FUNCTION_BLOCK EmergencyManagement (* CAT Function Block Type *)
  (* Standard: 61499-2 *)
  (* Version 0.0, 7/4/2026, Schneider Electric, template *)
  PACKAGE SE.Nereda;
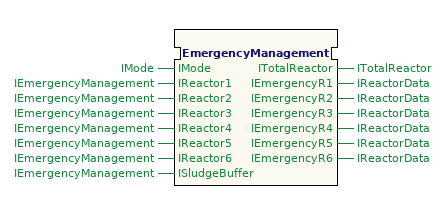
  SOCKETS
    IMode : IMode;
    IReactor1 : IEmergencyManagement;
    IReactor2 : IEmergencyManagement;
    IReactor3 : IEmergencyManagement;
    IReactor4 : IEmergencyManagement;
    IReactor5 : IEmergencyManagement;
    IReactor6 : IEmergencyManagement;
    ISludgeBuffer : IEmergencyManagement;
  END_SOCKETS
  PLUGS
    ITotalReactor : ITotalReactor;
    IEmergencyR1 : IReactorData(pin_7FC77B7D4B4A5A4D := 1);
    IEmergencyR2 : IReactorData(pin_7FC77B7D4B4A5A4D := 2);
    IEmergencyR3 : IReactorData(pin_7FC77B7D4B4A5A4D := 3);
    IEmergencyR4 : IReactorData(pin_7FC77B7D4B4A5A4D := 4);
    IEmergencyR5 : IReactorData(pin_7FC77B7D4B4A5A4D := 5);
    IEmergencyR6 : IReactorData(pin_7FC77B7D4B4A5A4D := 6);
  END_PLUGS
  (* 01 - FUNCTIONNAL INPUT INTERFACE *)
  (* 00 - INITIALIZATION *)
  (* 05 - LOGIC *)
  (* 06 - HMI INTERFACE *)
  (* 03 - FIELD INTERFACE *)
  (* 02 - FUNCTIONNAL OUTPUT INTERFACE *)
  (* Number of Reactors Exist *)
  (* 04 - CHILDREN *)
  (* 4A - TYPICALS *)
  (* Actual Cycle Time (CT_reactor_actual) CT_ReactorActual = (N_AvailableReactors / N_TotalReactors) x CT_Nominal *)
  (* Next Feed Horizon Calculation (Scheduler) *)
  (* Emergency ON *)
  (* Number of Reactors Available *)
  (* Start Feed Position *)
  (* Feed Interval (Start_IntervalV = CT_ReactorActual / N_AvailableReactors) *)
  (* Emergency Reactors Control (Start & Stop) *)
  (* Time Sice Start Feed *)
  (* Emergency Initialization *)
  (* Start Feed Position This functional block manages the reactor position order, which determines the sequence in which the feeds are started. We request an update of the "Reactor To Start Feed" position in the following two cases: - In the logic that controls the start of the Emergency Recipe Sequence. - In the update performed after the start of each feed. *)
  (* Comment These function blocks (`SD_WS2_Initialization_Manager` and `RxNoAvThenRxAv`) must be modified to match the number of reactors in your plant. *)
  FBS
    INIT : plcStart(Prio := 50, Delay := T#0ms);
    NumberOfReactors : ADD_196CF02D1C6422644; {SET_ATTRIBUTE(Configuration.GenericFBType.InterfaceParams, Runtime.Standard#CNT:=6;IN${CNT$}:LREAL)}
    IThis : EmergencyManagement_HMI(QI := TRUE);
    SmoothNumberOfReactors : LRealValueChanged;
    SmoothNumberOfReactors1 : LREAL2REAL;
    CT_ReactorActual : CT_ReactorActual;
    SmoothCT_ReactorActual : RealValueChanged;
    EmergencyON : COMPARE_739E3FB559152FE(IN2 := 3); {SET_ATTRIBUTE(Configuration.GenericFBType.InterfaceParams, Runtime.Standard#CNT:=2;IN${CNT$}:INT)}
    SmoothEmergencyON : boolValueChanged;
    NumberOfReactorsAv : ADD_196CF02D1C6422644; {SET_ATTRIBUTE(Configuration.GenericFBType.InterfaceParams, Runtime.Standard#CNT:=6;IN${CNT$}:LREAL)}
    SmoothNumberOfReactorsAv : LRealValueChanged;
    NumberOfReactorsAv2 : LREAL2REAL;
    BOOL2INT : BOOL2INT_6;
    StartFeedPosition : StartFeedPosition;
    SmoothNumberOfReactors2 : REAL2INT;
    ReactorFeedInterval : StartIntervalCalc;
    EmergencyReactorsControl : EmergencyManagementControl;
    NumberOfReactorsAv3 : REAL2INT;
    StartUpDelay : E_DELAY_V_D;
    Retrigger_StartFeedPosition : RetriggerEvent(pin_CFF51EFF0A91DC53 := 3, pin_FDD5DC24A8674AF6 := T#1s);
    ForceAvaibility : ReactorAvCtrl;
    SmoothFeedInterval : RealValueChanged;
    TimeSinceStartFeedR1 : RealValueChanged;
    TimeSinceStartFeedR2 : RealValueChanged;
    TimeSinceStartFeedR3 : RealValueChanged;
    TimeSinceStartFeedR4 : RealValueChanged;
    TimeSinceStartFeedR5 : RealValueChanged;
    TimeSinceStartFeedR6 : RealValueChanged;
    NextFeedHorizon : NextFeedHorizon;
    BOOL2INT1 : BOOL2INT_6;
    FeedRun : E_PERMIT;
    FeedStarted : OR_65BD917F4F2EC165; {SET_ATTRIBUTE(Configuration.GenericFBType.InterfaceParams, Runtime.Standard#CNT:=6;OUT:BOOL)}
    FeedCmdTimeOutR1 : TimeOut(pin_5F65B6CE2660F5EB := T#500ms);
    FeedCmdTimeOutR2 : TimeOut(pin_5F65B6CE2660F5EB := T#500ms);
    FeedCmdTimeOutR3 : TimeOut(pin_5F65B6CE2660F5EB := T#500ms);
    FeedCmdTimeOutR4 : TimeOut(pin_5F65B6CE2660F5EB := T#500ms);
    FeedCmdTimeOutR5 : TimeOut(pin_5F65B6CE2660F5EB := T#500ms);
    FeedCmdTimeOutR6 : TimeOut(pin_5F65B6CE2660F5EB := T#500ms);
    SD_WS2_Initialization_Manager : SDInitDone(pin_9BB0B293AF87503A := TRUE, pin_46B4EB9EBD3AAF12 := TRUE, pin_7A6A945A02239988 := TRUE);
    Wait : E_DELAY(DT := T#500ms);
    UPDATE_POS : E_DELAY(DT := T#1s);
    Delay : E_DELAY_V_D(DT1 := T#2s);
    FeedStartedSmooth : BoolValueChanged_6;
    ReactorAvaibilityChanged : BoolValueChanged_6;
    UPDATE_POS_EO : E_MERGE;
    EmergencyONPermit : E_PERMIT;
    RxNoAvThenRxAv : RNoAvThenRAv(pin_F258A2B490CD5DB0 := TRUE, pin_1987E369E19A00E5 := TRUE, pin_36BA10F8F7A678CF := TRUE);
    Wait1 : E_DELAY(DT := T#500ms);
  END_FBS
  EVENT_CONNECTIONS
    EmergencyON.CNF TO SmoothEmergencyON.REQ;
    IMode.MODE TO EmergencyON.REQ;
    IMode.MODE TO EmergencyReactorsControl.57E2081A00120193;
    IReactor2.PHASE_NO_ABORTED TO ForceAvaibility.AA8C7A967C5CED2A;
    IReactor2.PHASE_NO_ABORTED TO EmergencyReactorsControl.FC096638C9B2EBE7;
    IReactor2.FEED_TIME TO StartFeedPosition.9A3C6DCF3E2E1FB0;
    IReactor2.12FB600C11F75EA2 TO StartFeedPosition.9A3C6DCF3E2E1FB0;
    IReactor2.12FB600C11F75EA2 TO EmergencyReactorsControl.3FB25A98F6D2D397;
    IReactor2.12FB600C11F75EA2 TO EmergencyReactorsControl.FC096638C9B2EBE7;
    StartUpDelay.INITO TO IReactor2.33EC5B834E8FFAF3;
    IReactor1.PHASE_NO_ABORTED TO ForceAvaibility.AA8C7A967C5CED2A;
    IReactor1.PHASE_NO_ABORTED TO EmergencyReactorsControl.FC096638C9B2EBE7;
    IReactor1.FEED_TIME TO StartFeedPosition.9A3C6DCF3E2E1FB0;
    IReactor1.12FB600C11F75EA2 TO StartFeedPosition.9A3C6DCF3E2E1FB0;
    IReactor1.12FB600C11F75EA2 TO EmergencyReactorsControl.3FB25A98F6D2D397;
    IReactor1.12FB600C11F75EA2 TO EmergencyReactorsControl.FC096638C9B2EBE7;
    StartUpDelay.INITO TO IReactor1.33EC5B834E8FFAF3;
    StartUpDelay.INITO TO IReactor3.33EC5B834E8FFAF3;
    IReactor3.PHASE_NO_ABORTED TO ForceAvaibility.AA8C7A967C5CED2A;
    IReactor3.PHASE_NO_ABORTED TO EmergencyReactorsControl.FC096638C9B2EBE7;
    IReactor3.FEED_TIME TO StartFeedPosition.9A3C6DCF3E2E1FB0;
    IReactor3.12FB600C11F75EA2 TO StartFeedPosition.9A3C6DCF3E2E1FB0;
    IReactor3.12FB600C11F75EA2 TO EmergencyReactorsControl.3FB25A98F6D2D397;
    IReactor3.12FB600C11F75EA2 TO EmergencyReactorsControl.FC096638C9B2EBE7;
    StartUpDelay.INITO TO IReactor4.33EC5B834E8FFAF3;
    IReactor4.PHASE_NO_ABORTED TO ForceAvaibility.AA8C7A967C5CED2A;
    IReactor4.PHASE_NO_ABORTED TO EmergencyReactorsControl.FC096638C9B2EBE7;
    IReactor4.FEED_TIME TO StartFeedPosition.9A3C6DCF3E2E1FB0;
    IReactor4.12FB600C11F75EA2 TO StartFeedPosition.9A3C6DCF3E2E1FB0;
    IReactor4.12FB600C11F75EA2 TO EmergencyReactorsControl.3FB25A98F6D2D397;
    IReactor4.12FB600C11F75EA2 TO EmergencyReactorsControl.FC096638C9B2EBE7;
    StartUpDelay.INITO TO IReactor5.33EC5B834E8FFAF3;
    IReactor5.PHASE_NO_ABORTED TO ForceAvaibility.AA8C7A967C5CED2A;
    IReactor5.PHASE_NO_ABORTED TO EmergencyReactorsControl.FC096638C9B2EBE7;
    IReactor5.FEED_TIME TO StartFeedPosition.9A3C6DCF3E2E1FB0;
    IReactor5.12FB600C11F75EA2 TO StartFeedPosition.9A3C6DCF3E2E1FB0;
    IReactor5.12FB600C11F75EA2 TO EmergencyReactorsControl.3FB25A98F6D2D397;
    IReactor5.12FB600C11F75EA2 TO EmergencyReactorsControl.FC096638C9B2EBE7;
    IReactor6.PHASE_NO_ABORTED TO ForceAvaibility.AA8C7A967C5CED2A;
    IReactor6.PHASE_NO_ABORTED TO EmergencyReactorsControl.FC096638C9B2EBE7;
    IReactor6.FEED_TIME TO StartFeedPosition.9A3C6DCF3E2E1FB0;
    IReactor6.12FB600C11F75EA2 TO StartFeedPosition.9A3C6DCF3E2E1FB0;
    IReactor6.12FB600C11F75EA2 TO EmergencyReactorsControl.3FB25A98F6D2D397;
    IReactor6.12FB600C11F75EA2 TO EmergencyReactorsControl.FC096638C9B2EBE7;
    StartUpDelay.INITO TO IReactor6.33EC5B834E8FFAF3;
    SmoothNumberOfReactors2.6FC99A5BD1C38561 TO EmergencyReactorsControl.3FB25A98F6D2D397;
    NumberOfReactorsAv3.6FC99A5BD1C38561 TO EmergencyReactorsControl.FC096638C9B2EBE7;
    StartUpDelay.1457E63E0C241C83 TO EmergencyReactorsControl.B99EA0FFDDD9DD73;
    EmergencyReactorsControl.5425B5FF7C2B3EA7 TO IEmergencyR1.395F2A7D1AB6A478;
    EmergencyReactorsControl.5425B5FF7C2B3EA7 TO IEmergencyR2.395F2A7D1AB6A478;
    EmergencyReactorsControl.5425B5FF7C2B3EA7 TO IEmergencyR4.395F2A7D1AB6A478;
    EmergencyReactorsControl.5425B5FF7C2B3EA7 TO IEmergencyR3.395F2A7D1AB6A478;
    EmergencyReactorsControl.5425B5FF7C2B3EA7 TO IEmergencyR5.395F2A7D1AB6A478;
    EmergencyReactorsControl.5425B5FF7C2B3EA7 TO IEmergencyR6.395F2A7D1AB6A478;
    EmergencyReactorsControl.B331D681195361F6 TO StartUpDelay.START;
    StartUpDelay.INITO TO ForceAvaibility.227A3F3489EABE9B;
    SmoothNumberOfReactors2.6FC99A5BD1C38561 TO ITotalReactor.TOTAL_REACTOR;
    SmoothEmergencyON.CHD TO IEmergencyR1.E1D373823D64ACA0;
    SmoothEmergencyON.CHD TO IEmergencyR2.E1D373823D64ACA0;
    SmoothEmergencyON.CHD TO IEmergencyR3.E1D373823D64ACA0;
    SmoothEmergencyON.CHD TO IEmergencyR4.E1D373823D64ACA0;
    SmoothEmergencyON.CHD TO IEmergencyR5.E1D373823D64ACA0;
    SmoothEmergencyON.CHD TO IEmergencyR6.E1D373823D64ACA0;
    NumberOfReactors.CNF TO SmoothNumberOfReactors.77F8F9CFF707DAFF;
    SmoothNumberOfReactors.93AE3729A9342678 TO SmoothNumberOfReactors1.DD5870AA881150BB;
    SmoothNumberOfReactors1.6FC99A5BD1C38561 TO SmoothNumberOfReactors2.DD5870AA881150BB;
    SmoothNumberOfReactors2.6FC99A5BD1C38561 TO CT_ReactorActual.B5AD92DA165DFC02;
    BOOL2INT.6FC99A5BD1C38561 TO NumberOfReactorsAv.REQ;
    NumberOfReactorsAv.CNF TO SmoothNumberOfReactorsAv.77F8F9CFF707DAFF;
    SmoothNumberOfReactorsAv.93AE3729A9342678 TO NumberOfReactorsAv2.DD5870AA881150BB;
    NumberOfReactorsAv2.6FC99A5BD1C38561 TO NumberOfReactorsAv3.DD5870AA881150BB;
    NumberOfReactorsAv3.6FC99A5BD1C38561 TO CT_ReactorActual.B5AD92DA165DFC02;
    NumberOfReactorsAv3.6FC99A5BD1C38561 TO ReactorFeedInterval.56116EFC174D2765;
    CT_ReactorActual.FB6D4D448571E6B8 TO SmoothCT_ReactorActual.77F8F9CFF707DAFF;
    SmoothCT_ReactorActual.93AE3729A9342678 TO ReactorFeedInterval.56116EFC174D2765;
    EmergencyReactorsControl.4DD14AD6E2842102 TO StartFeedPosition.DD2DDDBAAA645E47;
    SmoothNumberOfReactorsAv.350834820611931F TO StartFeedPosition.9A3C6DCF3E2E1FB0;
    Retrigger_StartFeedPosition.4002AEF0814D09CF TO EmergencyReactorsControl.7CCC917F1D2D8CDF;
    SmoothCT_ReactorActual.93AE3729A9342678 TO IEmergencyR1.198EF041C70827BC;
    SmoothCT_ReactorActual.93AE3729A9342678 TO IEmergencyR2.198EF041C70827BC;
    SmoothCT_ReactorActual.93AE3729A9342678 TO IEmergencyR3.198EF041C70827BC;
    SmoothCT_ReactorActual.93AE3729A9342678 TO IEmergencyR4.198EF041C70827BC;
    SmoothCT_ReactorActual.93AE3729A9342678 TO IEmergencyR5.198EF041C70827BC;
    SmoothCT_ReactorActual.93AE3729A9342678 TO IEmergencyR6.198EF041C70827BC;
    SmoothFeedInterval.93AE3729A9342678 TO IEmergencyR1.9D1E5F7369C5538B;
    SmoothFeedInterval.93AE3729A9342678 TO IEmergencyR2.9D1E5F7369C5538B;
    SmoothFeedInterval.93AE3729A9342678 TO IEmergencyR3.9D1E5F7369C5538B;
    SmoothFeedInterval.93AE3729A9342678 TO IEmergencyR4.9D1E5F7369C5538B;
    SmoothFeedInterval.93AE3729A9342678 TO IEmergencyR5.9D1E5F7369C5538B;
    SmoothFeedInterval.93AE3729A9342678 TO IEmergencyR6.9D1E5F7369C5538B;
    EmergencyReactorsControl.E01285EC1A4C329B TO IEmergencyR1.61CD32E3E6AEDF7D;
    EmergencyReactorsControl.E01285EC1A4C329B TO IEmergencyR2.61CD32E3E6AEDF7D;
    EmergencyReactorsControl.E01285EC1A4C329B TO IEmergencyR3.61CD32E3E6AEDF7D;
    EmergencyReactorsControl.E01285EC1A4C329B TO IEmergencyR4.61CD32E3E6AEDF7D;
    EmergencyReactorsControl.E01285EC1A4C329B TO IEmergencyR5.61CD32E3E6AEDF7D;
    EmergencyReactorsControl.E01285EC1A4C329B TO IEmergencyR6.61CD32E3E6AEDF7D;
    Retrigger_StartFeedPosition.4002AEF0814D09CF TO IEmergencyR1.911F6EFE27823BFD;
    Retrigger_StartFeedPosition.4002AEF0814D09CF TO IEmergencyR2.911F6EFE27823BFD;
    Retrigger_StartFeedPosition.4002AEF0814D09CF TO IEmergencyR3.911F6EFE27823BFD;
    Retrigger_StartFeedPosition.4002AEF0814D09CF TO IEmergencyR4.911F6EFE27823BFD;
    Retrigger_StartFeedPosition.4002AEF0814D09CF TO IEmergencyR5.911F6EFE27823BFD;
    Retrigger_StartFeedPosition.4002AEF0814D09CF TO IEmergencyR6.911F6EFE27823BFD;
    ForceAvaibility.A1ADA5210E38DA8E TO BOOL2INT.DD5870AA881150BB;
    ForceAvaibility.8EE38BB13A892011 TO NextFeedHorizon.E161DD05340F6BD8;
    ReactorFeedInterval.8A437FBF24BFC92F TO SmoothFeedInterval.77F8F9CFF707DAFF;
    EmergencyReactorsControl.BDC96AACAB3D2769 TO IEmergencyR1.1C1DD8946F24CFF9;
    EmergencyReactorsControl.BDC96AACAB3D2769 TO IEmergencyR2.1C1DD8946F24CFF9;
    EmergencyReactorsControl.BDC96AACAB3D2769 TO IEmergencyR3.1C1DD8946F24CFF9;
    EmergencyReactorsControl.BDC96AACAB3D2769 TO IEmergencyR4.1C1DD8946F24CFF9;
    EmergencyReactorsControl.BDC96AACAB3D2769 TO IEmergencyR5.1C1DD8946F24CFF9;
    EmergencyReactorsControl.BDC96AACAB3D2769 TO IEmergencyR6.1C1DD8946F24CFF9;
    IReactor1.FEED_TIME TO TimeSinceStartFeedR1.77F8F9CFF707DAFF;
    IReactor2.FEED_TIME TO TimeSinceStartFeedR1.77F8F9CFF707DAFF;
    IReactor3.FEED_TIME TO TimeSinceStartFeedR1.77F8F9CFF707DAFF;
    IReactor4.FEED_TIME TO TimeSinceStartFeedR1.77F8F9CFF707DAFF;
    IReactor5.FEED_TIME TO TimeSinceStartFeedR1.77F8F9CFF707DAFF;
    IReactor6.FEED_TIME TO TimeSinceStartFeedR1.77F8F9CFF707DAFF;
    TimeSinceStartFeedR1.350834820611931F TO TimeSinceStartFeedR2.77F8F9CFF707DAFF;
    TimeSinceStartFeedR2.350834820611931F TO TimeSinceStartFeedR3.77F8F9CFF707DAFF;
    TimeSinceStartFeedR4.350834820611931F TO TimeSinceStartFeedR5.77F8F9CFF707DAFF;
    TimeSinceStartFeedR5.350834820611931F TO TimeSinceStartFeedR6.77F8F9CFF707DAFF;
    TimeSinceStartFeedR3.350834820611931F TO TimeSinceStartFeedR4.77F8F9CFF707DAFF;
    NextFeedHorizon.D6F8783AE30F537C TO Delay.INIT;
    SmoothFeedInterval.93AE3729A9342678 TO NextFeedHorizon.7F05D9AA837FB21B;
    TimeSinceStartFeedR1.93AE3729A9342678 TO NextFeedHorizon.7F05D9AA837FB21B;
    TimeSinceStartFeedR2.93AE3729A9342678 TO NextFeedHorizon.7F05D9AA837FB21B;
    TimeSinceStartFeedR3.93AE3729A9342678 TO NextFeedHorizon.7F05D9AA837FB21B;
    TimeSinceStartFeedR4.93AE3729A9342678 TO NextFeedHorizon.7F05D9AA837FB21B;
    TimeSinceStartFeedR5.93AE3729A9342678 TO NextFeedHorizon.7F05D9AA837FB21B;
    TimeSinceStartFeedR6.93AE3729A9342678 TO NextFeedHorizon.7F05D9AA837FB21B;
    Retrigger_StartFeedPosition.4002AEF0814D09CF TO NextFeedHorizon.7F05D9AA837FB21B;
    NumberOfReactorsAv3.6FC99A5BD1C38561 TO NextFeedHorizon.7F05D9AA837FB21B;
    SmoothNumberOfReactors2.6FC99A5BD1C38561 TO NextFeedHorizon.7F05D9AA837FB21B;
    IReactor1.12FB600C11F75EA2 TO BOOL2INT1.DD5870AA881150BB;
    IReactor2.12FB600C11F75EA2 TO BOOL2INT1.DD5870AA881150BB;
    IReactor3.12FB600C11F75EA2 TO BOOL2INT1.DD5870AA881150BB;
    IReactor4.12FB600C11F75EA2 TO BOOL2INT1.DD5870AA881150BB;
    IReactor5.12FB600C11F75EA2 TO BOOL2INT1.DD5870AA881150BB;
    IReactor6.12FB600C11F75EA2 TO BOOL2INT1.DD5870AA881150BB;
    BOOL2INT1.6FC99A5BD1C38561 TO NumberOfReactors.REQ;
    NextFeedHorizon.A8C1183CD65D2C2F TO EmergencyReactorsControl.F396AB99E066BF1B;
    NextFeedHorizon.3C658083FB00E376 TO EmergencyReactorsControl.EE2641E02BEB131E;
    ForceAvaibility.D789D01B8B35E207 TO IEmergencyR1.7D5F3067068DE334;
    ForceAvaibility.D789D01B8B35E207 TO IEmergencyR2.7D5F3067068DE334;
    ForceAvaibility.D789D01B8B35E207 TO IEmergencyR3.7D5F3067068DE334;
    ForceAvaibility.D789D01B8B35E207 TO IEmergencyR4.7D5F3067068DE334;
    ForceAvaibility.D789D01B8B35E207 TO IEmergencyR5.7D5F3067068DE334;
    ForceAvaibility.D789D01B8B35E207 TO IEmergencyR6.7D5F3067068DE334;
    INIT.FIRST_INIT TO IThis.11B0EEC0AF1F6F5A;
    INIT.REDO_INIT TO IThis.11B0EEC0AF1F6F5A;
    Retrigger_StartFeedPosition.4002AEF0814D09CF TO IThis.6A631B6723098E8B;
    IEmergencyR1.D499D06F1953A020 TO IThis.6A631B6723098E8B;
    IReactor1.FEED_TIME TO IThis.6A631B6723098E8B;
    Retrigger_StartFeedPosition.4002AEF0814D09CF TO IThis.662D34935A18D4C8;
    IEmergencyR2.D499D06F1953A020 TO IThis.662D34935A18D4C8;
    IReactor2.FEED_TIME TO IThis.662D34935A18D4C8;
    IReactor3.FEED_TIME TO IThis.D5FE897AB4BE07D5;
    Retrigger_StartFeedPosition.4002AEF0814D09CF TO IThis.D5FE897AB4BE07D5;
    IEmergencyR3.D499D06F1953A020 TO IThis.D5FE897AB4BE07D5;
    Retrigger_StartFeedPosition.4002AEF0814D09CF TO IThis.0FC97BC77AEF2FB1;
    IEmergencyR4.D499D06F1953A020 TO IThis.0FC97BC77AEF2FB1;
    Retrigger_StartFeedPosition.4002AEF0814D09CF TO IThis.AD50BDBEE1844666;
    IEmergencyR5.D499D06F1953A020 TO IThis.AD50BDBEE1844666;
    Retrigger_StartFeedPosition.4002AEF0814D09CF TO IThis.883D86C4850F1B98;
    IEmergencyR6.D499D06F1953A020 TO IThis.883D86C4850F1B98;
    SmoothCT_ReactorActual.93AE3729A9342678 TO IThis.BCC6AEC920D25E91;
    IThis.B3B324179F7F1286 TO IThis.6FE84D876AB4D285;
    SmoothNumberOfReactors2.6FC99A5BD1C38561 TO IThis.6FE84D876AB4D285;
    NumberOfReactorsAv3.6FC99A5BD1C38561 TO IThis.6FE84D876AB4D285;
    SmoothFeedInterval.93AE3729A9342678 TO IThis.FF5508DDAEC8BEFB;
    EmergencyReactorsControl.57B86B24E58CE6DD TO IThis.C9F34726889CA7BE;
    SmoothEmergencyON.CHD TO IThis.9D03013895CCEF05;
    StartUpDelay.INITO TO IThis.32376FF6F2E25CA6;
    IThis.69E91E9E46EEE4A5 TO StartUpDelay.INIT;
    IThis.B3B324179F7F1286 TO CT_ReactorActual.B5AD92DA165DFC02;
    IThis.13B659E2726FB2AF TO StartUpDelay.8C325F07198FCB13;
    IReactor4.FEED_TIME TO IThis.0FC97BC77AEF2FB1;
    IReactor5.FEED_TIME TO IThis.AD50BDBEE1844666;
    IReactor6.FEED_TIME TO IThis.883D86C4850F1B98;
    NextFeedHorizon.5939463105CA5EBC TO IEmergencyR1.B3BDDBF095B97A2B;
    NextFeedHorizon.5939463105CA5EBC TO IEmergencyR2.B3BDDBF095B97A2B;
    NextFeedHorizon.5939463105CA5EBC TO IEmergencyR3.B3BDDBF095B97A2B;
    NextFeedHorizon.5939463105CA5EBC TO IEmergencyR4.B3BDDBF095B97A2B;
    NextFeedHorizon.5939463105CA5EBC TO IEmergencyR5.B3BDDBF095B97A2B;
    NextFeedHorizon.5939463105CA5EBC TO IEmergencyR6.B3BDDBF095B97A2B;
    FeedStarted.CNF TO FeedRun.EI;
    IEmergencyR1.138EEC247A2C05E7 TO FeedStartedSmooth.77F8F9CFF707DAFF;
    IEmergencyR2.138EEC247A2C05E7 TO FeedStartedSmooth.77F8F9CFF707DAFF;
    IEmergencyR3.138EEC247A2C05E7 TO FeedStartedSmooth.77F8F9CFF707DAFF;
    IEmergencyR4.138EEC247A2C05E7 TO FeedStartedSmooth.77F8F9CFF707DAFF;
    IEmergencyR5.138EEC247A2C05E7 TO FeedStartedSmooth.77F8F9CFF707DAFF;
    IEmergencyR6.138EEC247A2C05E7 TO FeedStartedSmooth.77F8F9CFF707DAFF;
    EmergencyReactorsControl.6CCD34FECBD70B12 TO StartUpDelay.STOP;
    FeedCmdTimeOutR1.A86E94B0584B0184 TO IEmergencyR1.395F2A7D1AB6A478;
    FeedCmdTimeOutR2.A86E94B0584B0184 TO IEmergencyR2.395F2A7D1AB6A478;
    FeedCmdTimeOutR3.A86E94B0584B0184 TO IEmergencyR3.395F2A7D1AB6A478;
    FeedCmdTimeOutR4.A86E94B0584B0184 TO IEmergencyR4.395F2A7D1AB6A478;
    FeedCmdTimeOutR5.A86E94B0584B0184 TO IEmergencyR5.395F2A7D1AB6A478;
    FeedCmdTimeOutR6.A86E94B0584B0184 TO IEmergencyR6.395F2A7D1AB6A478;
    EmergencyReactorsControl.5425B5FF7C2B3EA7 TO FeedCmdTimeOutR1.C17BD4ED345C3B34;
    EmergencyReactorsControl.5425B5FF7C2B3EA7 TO FeedCmdTimeOutR2.C17BD4ED345C3B34;
    EmergencyReactorsControl.5425B5FF7C2B3EA7 TO FeedCmdTimeOutR3.C17BD4ED345C3B34;
    EmergencyReactorsControl.5425B5FF7C2B3EA7 TO FeedCmdTimeOutR4.C17BD4ED345C3B34;
    EmergencyReactorsControl.5425B5FF7C2B3EA7 TO FeedCmdTimeOutR5.C17BD4ED345C3B34;
    EmergencyReactorsControl.5425B5FF7C2B3EA7 TO FeedCmdTimeOutR6.C17BD4ED345C3B34;
    IEmergencyR1.138EEC247A2C05E7 TO FeedCmdTimeOutR1.99EC5987D752BADB;
    IEmergencyR2.138EEC247A2C05E7 TO FeedCmdTimeOutR2.99EC5987D752BADB;
    IEmergencyR3.138EEC247A2C05E7 TO FeedCmdTimeOutR3.99EC5987D752BADB;
    IEmergencyR4.138EEC247A2C05E7 TO FeedCmdTimeOutR4.99EC5987D752BADB;
    IEmergencyR5.138EEC247A2C05E7 TO FeedCmdTimeOutR5.99EC5987D752BADB;
    IEmergencyR6.138EEC247A2C05E7 TO FeedCmdTimeOutR6.99EC5987D752BADB;
    NextFeedHorizon.D6F8783AE30F537C TO IEmergencyR1.CF316F4BA7C11A07;
    NextFeedHorizon.D6F8783AE30F537C TO IEmergencyR2.CF316F4BA7C11A07;
    NextFeedHorizon.D6F8783AE30F537C TO IEmergencyR3.CF316F4BA7C11A07;
    NextFeedHorizon.D6F8783AE30F537C TO IEmergencyR4.CF316F4BA7C11A07;
    NextFeedHorizon.D6F8783AE30F537C TO IEmergencyR5.CF316F4BA7C11A07;
    NextFeedHorizon.D6F8783AE30F537C TO IEmergencyR6.CF316F4BA7C11A07;
    EmergencyReactorsControl.E01285EC1A4C329B TO SD_WS2_Initialization_Manager.B4ABE90B67562793;
    SmoothEmergencyON.CHD TO SD_WS2_Initialization_Manager.08F744362D65AFEF;
    SD_WS2_Initialization_Manager.349B3D6587A5C960 TO IEmergencyR1.77175193A5DFB16A;
    SD_WS2_Initialization_Manager.349B3D6587A5C960 TO IEmergencyR2.77175193A5DFB16A;
    SD_WS2_Initialization_Manager.349B3D6587A5C960 TO IEmergencyR3.77175193A5DFB16A;
    SD_WS2_Initialization_Manager.349B3D6587A5C960 TO IEmergencyR4.77175193A5DFB16A;
    SD_WS2_Initialization_Manager.349B3D6587A5C960 TO IEmergencyR5.77175193A5DFB16A;
    SD_WS2_Initialization_Manager.349B3D6587A5C960 TO IEmergencyR6.77175193A5DFB16A;
    SD_WS2_Initialization_Manager.EE5D157431DCAF03 TO Wait.START;
    Wait.EO TO SD_WS2_Initialization_Manager.D6BB3A31A896D022;
    IEmergencyR1.48081868B719DABE TO SD_WS2_Initialization_Manager.161A69C360740A5D;
    IEmergencyR2.48081868B719DABE TO SD_WS2_Initialization_Manager.161A69C360740A5D;
    IEmergencyR3.48081868B719DABE TO SD_WS2_Initialization_Manager.161A69C360740A5D;
    IEmergencyR4.48081868B719DABE TO SD_WS2_Initialization_Manager.161A69C360740A5D;
    IEmergencyR5.48081868B719DABE TO SD_WS2_Initialization_Manager.161A69C360740A5D;
    IEmergencyR6.48081868B719DABE TO SD_WS2_Initialization_Manager.161A69C360740A5D;
    NextFeedHorizon.6B401466A075E8D5 TO EmergencyReactorsControl.CAB3BCEC18441220;
    FeedRun.EO TO UPDATE_POS_EO.EI1;
    UPDATE_POS.EO TO StartFeedPosition.DD2DDDBAAA645E47;
    StartFeedPosition.0BBB611D4A1D02F5 TO Retrigger_StartFeedPosition.2BC1963D96179493;
    Delay.INITO TO INIT.ACK_FIRST;
    SD_WS2_Initialization_Manager.61969B4370714317 TO Delay.START;
    SD_WS2_Initialization_Manager.965A154310F12DA0 TO Delay.STOP;
    Delay.1457E63E0C241C83 TO SD_WS2_Initialization_Manager.C1672E927894D208;
    SmoothEmergencyON.CHD TO StartFeedPosition.9A3C6DCF3E2E1FB0;
    SmoothNumberOfReactors2.6FC99A5BD1C38561 TO StartFeedPosition.9A3C6DCF3E2E1FB0;
    NumberOfReactorsAv3.6FC99A5BD1C38561 TO StartFeedPosition.9A3C6DCF3E2E1FB0;
    FeedStartedSmooth.93AE3729A9342678 TO FeedStarted.REQ;
    IReactor1.PHASE_NO_ABORTED TO ReactorAvaibilityChanged.77F8F9CFF707DAFF;
    IReactor2.PHASE_NO_ABORTED TO ReactorAvaibilityChanged.77F8F9CFF707DAFF;
    IReactor3.PHASE_NO_ABORTED TO ReactorAvaibilityChanged.77F8F9CFF707DAFF;
    IReactor4.PHASE_NO_ABORTED TO ReactorAvaibilityChanged.77F8F9CFF707DAFF;
    IReactor5.PHASE_NO_ABORTED TO ReactorAvaibilityChanged.77F8F9CFF707DAFF;
    IReactor6.PHASE_NO_ABORTED TO ReactorAvaibilityChanged.77F8F9CFF707DAFF;
    EmergencyONPermit.EO TO UPDATE_POS_EO.EI2;
    UPDATE_POS_EO.EO TO UPDATE_POS.START;
    ReactorAvaibilityChanged.93AE3729A9342678 TO EmergencyONPermit.EI;
    RxNoAvThenRxAv.36C8FEB2AEE2D77A TO Wait1.START;
    Wait1.EO TO RxNoAvThenRxAv.2DB21E5C040C7006;
    ReactorAvaibilityChanged.93AE3729A9342678 TO RxNoAvThenRxAv.D34CB04DF38A6DEF;
    SmoothEmergencyON.CHD TO RxNoAvThenRxAv.D34CB04DF38A6DEF;
    RxNoAvThenRxAv.CDE3D6C9BB9E2A16 TO IEmergencyR1.61CD32E3E6AEDF7D;
    RxNoAvThenRxAv.CDE3D6C9BB9E2A16 TO IEmergencyR2.61CD32E3E6AEDF7D;
    RxNoAvThenRxAv.CDE3D6C9BB9E2A16 TO IEmergencyR3.61CD32E3E6AEDF7D;
    RxNoAvThenRxAv.CDE3D6C9BB9E2A16 TO IEmergencyR4.61CD32E3E6AEDF7D;
    RxNoAvThenRxAv.CDE3D6C9BB9E2A16 TO IEmergencyR5.61CD32E3E6AEDF7D;
    RxNoAvThenRxAv.CDE3D6C9BB9E2A16 TO IEmergencyR6.61CD32E3E6AEDF7D;
    ISludgeBuffer.PHASE_NO_ABORTED TO IEmergencyR1.93812D9FEC4294F9;
    ISludgeBuffer.PHASE_NO_ABORTED TO IEmergencyR2.93812D9FEC4294F9;
    ISludgeBuffer.PHASE_NO_ABORTED TO IEmergencyR4.93812D9FEC4294F9;
    ISludgeBuffer.PHASE_NO_ABORTED TO IEmergencyR3.93812D9FEC4294F9;
    ISludgeBuffer.PHASE_NO_ABORTED TO IEmergencyR5.93812D9FEC4294F9;
    ISludgeBuffer.PHASE_NO_ABORTED TO IEmergencyR6.93812D9FEC4294F9;
  END_CONNECTIONS
  DATA_CONNECTIONS
    EmergencyON.EQ TO SmoothEmergencyON.Input;
    IMode.Mode TO EmergencyON.IN1;
    IMode.Mode TO EmergencyReactorsControl.E5B9CCCEF6B4EF65;
    IReactor2.3C69BB1A066E9338 TO ForceAvaibility.E2886DCF5F67CC3C;
    IReactor2.3C69BB1A066E9338 TO EmergencyReactorsControl.C849680A4A15ED1B;
    IReactor2.8FB3B1E89F73B5E3 TO StartFeedPosition.F6C5EC3F29BFB0F1;
    IReactor2.D997CA5474076632 TO StartFeedPosition.F243334218AD8632;
    IReactor2.D997CA5474076632 TO EmergencyReactorsControl.17A6E890A1D7837D;
    IReactor1.3C69BB1A066E9338 TO ForceAvaibility.7AD00457211990B7;
    IReactor1.3C69BB1A066E9338 TO EmergencyReactorsControl.EE41DCB738F42288;
    IReactor1.8FB3B1E89F73B5E3 TO StartFeedPosition.8F8E40FFA1871A34;
    IReactor1.D997CA5474076632 TO StartFeedPosition.2288C6CFF23884C8;
    IReactor1.D997CA5474076632 TO EmergencyReactorsControl.D64758C1D02B0BCD;
    IReactor3.3C69BB1A066E9338 TO ForceAvaibility.184AF3EDDA902CEB;
    IReactor3.3C69BB1A066E9338 TO EmergencyReactorsControl.5EDA85A673D3FE33;
    IReactor3.8FB3B1E89F73B5E3 TO StartFeedPosition.79B28AD4B979DF84;
    IReactor3.D997CA5474076632 TO StartFeedPosition.F86ECFC3CE58448E;
    IReactor3.D997CA5474076632 TO EmergencyReactorsControl.EA4BE6EBBFCF5C8B;
    IReactor4.3C69BB1A066E9338 TO ForceAvaibility.D8BF2694CDFF6342;
    IReactor4.3C69BB1A066E9338 TO EmergencyReactorsControl.457B120F292EA16A;
    IReactor4.8FB3B1E89F73B5E3 TO StartFeedPosition.C5DE4190999F922C;
    IReactor4.D997CA5474076632 TO StartFeedPosition.FB7CC18C7054818F;
    IReactor4.D997CA5474076632 TO EmergencyReactorsControl.DCC24ED92AA64397;
    IReactor5.3C69BB1A066E9338 TO ForceAvaibility.35342051FFEFD274;
    IReactor5.3C69BB1A066E9338 TO EmergencyReactorsControl.6537F2DBBFA180D6;
    IReactor5.8FB3B1E89F73B5E3 TO StartFeedPosition.45C5BFE5307DB06C;
    IReactor5.D997CA5474076632 TO StartFeedPosition.3A68F1D6CA6574E7;
    IReactor5.D997CA5474076632 TO EmergencyReactorsControl.0A25F1413330ACCE;
    IReactor6.3C69BB1A066E9338 TO ForceAvaibility.B952C03EAF905B1B;
    IReactor6.3C69BB1A066E9338 TO EmergencyReactorsControl.9520E907CE8A0D0D;
    IReactor6.8FB3B1E89F73B5E3 TO StartFeedPosition.299B36949DCFCE22;
    IReactor6.D997CA5474076632 TO StartFeedPosition.2179DB7FB0E14A2C;
    IReactor6.D997CA5474076632 TO EmergencyReactorsControl.17E973AAA9DB5F73;
    SmoothNumberOfReactors2.A6DEF5F9C27C1848 TO EmergencyReactorsControl.44C8149C8813B920;
    NumberOfReactorsAv3.A6DEF5F9C27C1848 TO EmergencyReactorsControl.87AC9CEF81AABFE3;
    StartFeedPosition.01DB13D42D3DBB3B TO EmergencyReactorsControl.7970D3D551982C0A;
    StartFeedPosition.6075D515D2693EEC TO EmergencyReactorsControl.268538F7EEE0D11C;
    StartFeedPosition.AE942E19AA2B17CE TO EmergencyReactorsControl.D608D5E19ABA04C1;
    StartFeedPosition.A0ADA3770331F35E TO EmergencyReactorsControl.66F3C3F6FFCC791F;
    StartFeedPosition.5073F46956E92D6C TO EmergencyReactorsControl.F1F69A85E585DE8B;
    StartFeedPosition.6BF52B2208BA01D0 TO EmergencyReactorsControl.CDE276592E415EA7;
    EmergencyReactorsControl.93BD970A79F50FF2 TO IEmergencyR1.B1FC30AB336AE8E9;
    EmergencyReactorsControl.48471A9871450B3D TO IEmergencyR2.B1FC30AB336AE8E9;
    EmergencyReactorsControl.C47F108F9D450515 TO IEmergencyR3.B1FC30AB336AE8E9;
    EmergencyReactorsControl.59886E5EA0464B37 TO IEmergencyR4.B1FC30AB336AE8E9;
    EmergencyReactorsControl.98828EA78D316628 TO IEmergencyR5.B1FC30AB336AE8E9;
    EmergencyReactorsControl.D66C5C5D632E05FA TO IEmergencyR6.B1FC30AB336AE8E9;
    SmoothNumberOfReactors1.A6DEF5F9C27C1848 TO ITotalReactor.TotalReactor;
    SmoothEmergencyON.Output TO IEmergencyR1.F0BEEA13B7FB6780;
    SmoothEmergencyON.Output TO IEmergencyR2.F0BEEA13B7FB6780;
    SmoothEmergencyON.Output TO IEmergencyR3.F0BEEA13B7FB6780;
    SmoothEmergencyON.Output TO IEmergencyR4.F0BEEA13B7FB6780;
    SmoothEmergencyON.Output TO IEmergencyR5.F0BEEA13B7FB6780;
    SmoothEmergencyON.Output TO IEmergencyR6.F0BEEA13B7FB6780;
    NumberOfReactors.OUT TO SmoothNumberOfReactors.25B5287A5784F3EC;
    SmoothNumberOfReactors.AA81B8787A42C5C8 TO SmoothNumberOfReactors1.4573FC8F228EB71D;
    SmoothNumberOfReactors1.A6DEF5F9C27C1848 TO SmoothNumberOfReactors2.4573FC8F228EB71D;
    BOOL2INT.A6DEF5F9C27C1848 TO NumberOfReactorsAv.IN1;
    BOOL2INT.515A2E3BB78F58C7 TO NumberOfReactorsAv.IN2;
    BOOL2INT.FCA64FB4B13F606F TO NumberOfReactorsAv.IN3;
    BOOL2INT.740A810221DABFBE TO NumberOfReactorsAv.IN4;
    BOOL2INT.E26587EB8B52B240 TO NumberOfReactorsAv.IN5;
    BOOL2INT.CC0A00FA21FBDB4C TO NumberOfReactorsAv.IN6;
    NumberOfReactorsAv.OUT TO SmoothNumberOfReactorsAv.25B5287A5784F3EC;
    SmoothNumberOfReactorsAv.AA81B8787A42C5C8 TO NumberOfReactorsAv2.4573FC8F228EB71D;
    NumberOfReactorsAv2.A6DEF5F9C27C1848 TO NumberOfReactorsAv3.4573FC8F228EB71D;
    NumberOfReactorsAv2.A6DEF5F9C27C1848 TO CT_ReactorActual.D315DE00E27AAC37;
    NumberOfReactorsAv2.A6DEF5F9C27C1848 TO ReactorFeedInterval.717B6E593DE7C489;
    CT_ReactorActual.C0B48C47E5E2C765 TO SmoothCT_ReactorActual.25B5287A5784F3EC;
    SmoothNumberOfReactors1.A6DEF5F9C27C1848 TO CT_ReactorActual.5E724B45B393A5A5;
    SmoothCT_ReactorActual.AA81B8787A42C5C8 TO ReactorFeedInterval.232FB5D2DFB3AE51;
    IReactor1.3C69BB1A066E9338 TO StartFeedPosition.DAD9CD3145CA8538;
    IReactor2.3C69BB1A066E9338 TO StartFeedPosition.487444B3AF9098A4;
    IReactor3.3C69BB1A066E9338 TO StartFeedPosition.E00536C09B387ACD;
    IReactor4.3C69BB1A066E9338 TO StartFeedPosition.C85115F3F80967FC;
    IReactor5.3C69BB1A066E9338 TO StartFeedPosition.8FC0347060032564;
    IReactor6.3C69BB1A066E9338 TO StartFeedPosition.88B5DA99424068DF;
    SmoothCT_ReactorActual.AA81B8787A42C5C8 TO IEmergencyR1.758E7E3A994DF6A3;
    SmoothCT_ReactorActual.AA81B8787A42C5C8 TO IEmergencyR2.758E7E3A994DF6A3;
    SmoothCT_ReactorActual.AA81B8787A42C5C8 TO IEmergencyR3.758E7E3A994DF6A3;
    SmoothCT_ReactorActual.AA81B8787A42C5C8 TO IEmergencyR4.758E7E3A994DF6A3;
    SmoothCT_ReactorActual.AA81B8787A42C5C8 TO IEmergencyR5.758E7E3A994DF6A3;
    SmoothCT_ReactorActual.AA81B8787A42C5C8 TO IEmergencyR6.758E7E3A994DF6A3;
    ReactorFeedInterval.6A936F9AECB0F130 TO IEmergencyR1.852A82A24B95110C;
    ReactorFeedInterval.6A936F9AECB0F130 TO IEmergencyR2.852A82A24B95110C;
    ReactorFeedInterval.6A936F9AECB0F130 TO IEmergencyR3.852A82A24B95110C;
    ReactorFeedInterval.6A936F9AECB0F130 TO IEmergencyR4.852A82A24B95110C;
    ReactorFeedInterval.6A936F9AECB0F130 TO IEmergencyR5.852A82A24B95110C;
    ReactorFeedInterval.6A936F9AECB0F130 TO IEmergencyR6.852A82A24B95110C;
    SmoothFeedInterval.AA81B8787A42C5C8 TO IEmergencyR1.7614E537E01F969F;
    SmoothFeedInterval.AA81B8787A42C5C8 TO IEmergencyR2.7614E537E01F969F;
    SmoothFeedInterval.AA81B8787A42C5C8 TO IEmergencyR3.7614E537E01F969F;
    SmoothFeedInterval.AA81B8787A42C5C8 TO IEmergencyR4.7614E537E01F969F;
    SmoothFeedInterval.AA81B8787A42C5C8 TO IEmergencyR5.7614E537E01F969F;
    SmoothFeedInterval.AA81B8787A42C5C8 TO IEmergencyR6.7614E537E01F969F;
    StartFeedPosition.01DB13D42D3DBB3B TO IEmergencyR1.074948F0B024FF2E;
    StartFeedPosition.6075D515D2693EEC TO IEmergencyR2.074948F0B024FF2E;
    StartFeedPosition.AE942E19AA2B17CE TO IEmergencyR3.074948F0B024FF2E;
    StartFeedPosition.A0ADA3770331F35E TO IEmergencyR4.074948F0B024FF2E;
    StartFeedPosition.5073F46956E92D6C TO IEmergencyR5.074948F0B024FF2E;
    StartFeedPosition.6BF52B2208BA01D0 TO IEmergencyR6.074948F0B024FF2E;
    ForceAvaibility.F22BC22150974352 TO BOOL2INT.4573FC8F228EB71D;
    ForceAvaibility.3C4B304BEF86E8FF TO BOOL2INT.DF8224FEB3446E92;
    ForceAvaibility.B101E63CA1FE77AB TO BOOL2INT.F547CEFAFDE5D422;
    ForceAvaibility.00225622EB9EF480 TO BOOL2INT.25941BC08BA9FF7D;
    ForceAvaibility.8177CB32FDF96C7A TO BOOL2INT.0FBE3E40D32297B2;
    ForceAvaibility.94CC84328D15AD2D TO BOOL2INT.D3CE592CD38CCBE1;
    ReactorFeedInterval.6C899D1F13E17AE7 TO SmoothFeedInterval.25B5287A5784F3EC;
    IReactor1.8FB3B1E89F73B5E3 TO TimeSinceStartFeedR1.25B5287A5784F3EC;
    IReactor2.8FB3B1E89F73B5E3 TO TimeSinceStartFeedR2.25B5287A5784F3EC;
    IReactor3.8FB3B1E89F73B5E3 TO TimeSinceStartFeedR3.25B5287A5784F3EC;
    IReactor4.8FB3B1E89F73B5E3 TO TimeSinceStartFeedR4.25B5287A5784F3EC;
    IReactor5.8FB3B1E89F73B5E3 TO TimeSinceStartFeedR5.25B5287A5784F3EC;
    IReactor6.8FB3B1E89F73B5E3 TO TimeSinceStartFeedR6.25B5287A5784F3EC;
    SmoothFeedInterval.AA81B8787A42C5C8 TO NextFeedHorizon.DAD5121B209FA0D7;
    TimeSinceStartFeedR1.AA81B8787A42C5C8 TO NextFeedHorizon.AEF7CA9732FE11A5;
    TimeSinceStartFeedR2.AA81B8787A42C5C8 TO NextFeedHorizon.5E5AE4C3F312A76B;
    TimeSinceStartFeedR3.AA81B8787A42C5C8 TO NextFeedHorizon.8DF2F6F4419686E2;
    TimeSinceStartFeedR4.AA81B8787A42C5C8 TO NextFeedHorizon.4B40AA2397BD41E8;
    TimeSinceStartFeedR5.AA81B8787A42C5C8 TO NextFeedHorizon.D7429B1EE301CDFE;
    TimeSinceStartFeedR6.AA81B8787A42C5C8 TO NextFeedHorizon.93F444735AD5D04C;
    StartFeedPosition.01DB13D42D3DBB3B TO NextFeedHorizon.5ED2D6B4B8E2C81B;
    StartFeedPosition.6075D515D2693EEC TO NextFeedHorizon.BD5E7F9FA8975C3D;
    StartFeedPosition.AE942E19AA2B17CE TO NextFeedHorizon.7B595B7E09BFF108;
    StartFeedPosition.A0ADA3770331F35E TO NextFeedHorizon.3D5EEF71869AC9D7;
    StartFeedPosition.5073F46956E92D6C TO NextFeedHorizon.AE40E4C82BF8C7E7;
    StartFeedPosition.6BF52B2208BA01D0 TO NextFeedHorizon.7DDD6AC011B3DBCD;
    IReactor1.D997CA5474076632 TO BOOL2INT1.4573FC8F228EB71D;
    IReactor2.D997CA5474076632 TO BOOL2INT1.DF8224FEB3446E92;
    BOOL2INT1.A6DEF5F9C27C1848 TO NumberOfReactors.IN1;
    BOOL2INT1.515A2E3BB78F58C7 TO NumberOfReactors.IN2;
    BOOL2INT1.FCA64FB4B13F606F TO NumberOfReactors.IN3;
    BOOL2INT1.740A810221DABFBE TO NumberOfReactors.IN4;
    BOOL2INT1.E26587EB8B52B240 TO NumberOfReactors.IN5;
    BOOL2INT1.CC0A00FA21FBDB4C TO NumberOfReactors.IN6;
    IReactor3.D997CA5474076632 TO BOOL2INT1.F547CEFAFDE5D422;
    IReactor4.D997CA5474076632 TO BOOL2INT1.25941BC08BA9FF7D;
    IReactor5.D997CA5474076632 TO BOOL2INT1.0FBE3E40D32297B2;
    IReactor6.D997CA5474076632 TO BOOL2INT1.D3CE592CD38CCBE1;
    IReactor1.D997CA5474076632 TO NextFeedHorizon.CDA279841963E2B6;
    IReactor2.D997CA5474076632 TO NextFeedHorizon.685F1999EF689540;
    IReactor3.D997CA5474076632 TO NextFeedHorizon.2B3B31727B3747FC;
    IReactor4.D997CA5474076632 TO NextFeedHorizon.546E546589B5351D;
    IReactor5.D997CA5474076632 TO NextFeedHorizon.6CE427190E7440DE;
    IReactor6.D997CA5474076632 TO NextFeedHorizon.6D4F67D2B423227C;
    IReactor1.3C69BB1A066E9338 TO NextFeedHorizon.56EE24DAF84918FB;
    IReactor2.3C69BB1A066E9338 TO NextFeedHorizon.F4328F61086BC2F2;
    IReactor3.3C69BB1A066E9338 TO NextFeedHorizon.38E1A69058BEFEAC;
    IReactor4.3C69BB1A066E9338 TO NextFeedHorizon.0418A012423811CE;
    IReactor5.3C69BB1A066E9338 TO NextFeedHorizon.DDA090357554230F;
    IReactor6.3C69BB1A066E9338 TO NextFeedHorizon.02C018DD15D9E328;
    NextFeedHorizon.AB599B0F98985E4C TO EmergencyReactorsControl.87691FC4DEA46E18;
    NextFeedHorizon.5CE4E81C12BD5FEE TO EmergencyReactorsControl.9BAC5A94B9B65D61;
    NextFeedHorizon.DC202AAF88E1AEA0 TO EmergencyReactorsControl.D86A2D3443DE924B;
    NextFeedHorizon.1E52C913E4BF284D TO EmergencyReactorsControl.712924DB38A0094F;
    NextFeedHorizon.1A9BCC64380D58EB TO EmergencyReactorsControl.3F0EC98BBFEFD461;
    NextFeedHorizon.2E490A1F4619D2A5 TO EmergencyReactorsControl.4CC5F004B67ABC18;
    EmergencyReactorsControl.27C27D9D7E3A4C1B TO IEmergencyR1.3C27B3AC98B413B4;
    CT_ReactorActual.D87066B84ABC3E2B TO IEmergencyR5.90388C221FF11A3D;
    CT_ReactorActual.D87066B84ABC3E2B TO IEmergencyR6.90388C221FF11A3D;
    CT_ReactorActual.D87066B84ABC3E2B TO IEmergencyR3.90388C221FF11A3D;
    CT_ReactorActual.D87066B84ABC3E2B TO IEmergencyR4.90388C221FF11A3D;
    CT_ReactorActual.D87066B84ABC3E2B TO IEmergencyR2.90388C221FF11A3D;
    CT_ReactorActual.D87066B84ABC3E2B TO IEmergencyR1.90388C221FF11A3D;
    EmergencyReactorsControl.27C27D9D7E3A4C1B TO IEmergencyR2.3C27B3AC98B413B4;
    EmergencyReactorsControl.27C27D9D7E3A4C1B TO IEmergencyR3.3C27B3AC98B413B4;
    EmergencyReactorsControl.27C27D9D7E3A4C1B TO IEmergencyR4.3C27B3AC98B413B4;
    EmergencyReactorsControl.27C27D9D7E3A4C1B TO IEmergencyR5.3C27B3AC98B413B4;
    EmergencyReactorsControl.27C27D9D7E3A4C1B TO IEmergencyR6.3C27B3AC98B413B4;
    NextFeedHorizon.F15D4AB48B43B912 TO EmergencyReactorsControl.E3F1DE02F9D441C1;
    NextFeedHorizon.E23396371F0D8536 TO EmergencyReactorsControl.425978B4225D5A81;
    ForceAvaibility.A23A844C33390AC2 TO IEmergencyR1.35F3027F47B7A966;
    ForceAvaibility.CE96517891BAC0E7 TO IEmergencyR2.35F3027F47B7A966;
    ForceAvaibility.BC4BA27376CCB235 TO IEmergencyR3.35F3027F47B7A966;
    ForceAvaibility.61AAEC2D50AC09D5 TO IEmergencyR4.35F3027F47B7A966;
    ForceAvaibility.FEDB450F513CB826 TO IEmergencyR5.35F3027F47B7A966;
    ForceAvaibility.8256E9C92E0FD34E TO IEmergencyR6.35F3027F47B7A966;
    IReactor1.B60AD268A06073AC TO IThis.B63CDC12742BD7C7;
    IEmergencyR1.793E1D04BE895F4E TO IThis.3D5D7029E013F5C3;
    StartFeedPosition.01DB13D42D3DBB3B TO IThis.42B41E72FF116C49;
    IReactor2.B60AD268A06073AC TO IThis.006BCC1F28671540;
    IEmergencyR2.793E1D04BE895F4E TO IThis.C541550A7B8396B6;
    StartFeedPosition.6075D515D2693EEC TO IThis.14BFB9EC5D11BAC0;
    IReactor3.B60AD268A06073AC TO IThis.5AF103287BB6082F;
    IEmergencyR3.793E1D04BE895F4E TO IThis.3A221D9ECFCDD8E8;
    StartFeedPosition.AE942E19AA2B17CE TO IThis.8CA933C146CE004C;
    IReactor4.B60AD268A06073AC TO IThis.ED873C8DD82E6926;
    IEmergencyR4.793E1D04BE895F4E TO IThis.D7259444B3D53457;
    StartFeedPosition.A0ADA3770331F35E TO IThis.A74D0C5FA39EF1A7;
    IReactor5.B60AD268A06073AC TO IThis.F3B989653CB07C14;
    IEmergencyR5.793E1D04BE895F4E TO IThis.A1624FC2D318C921;
    StartFeedPosition.5073F46956E92D6C TO IThis.4DE93E0CD3748B9A;
    IReactor6.B60AD268A06073AC TO IThis.9F10D13CD9C7C018;
    IEmergencyR6.793E1D04BE895F4E TO IThis.78C911374139C4A5;
    StartFeedPosition.6BF52B2208BA01D0 TO IThis.FE6B4FE46513E874;
    CT_ReactorActual.D87066B84ABC3E2B TO IThis.5FCE4BE5D3541CF3;
    SmoothNumberOfReactors2.A6DEF5F9C27C1848 TO IThis.10AAE963FE9CCB49;
    NumberOfReactorsAv3.A6DEF5F9C27C1848 TO IThis.77E421A3AAD17708;
    IThis.90008E8CE94947BC TO IThis.C41E2CBE27C99742;
    ReactorFeedInterval.6A936F9AECB0F130 TO IThis.55813B244AB7A7F6;
    EmergencyReactorsControl.8BF438286778ED88 TO IThis.7BAB8EF95999CA3E;
    SmoothEmergencyON.Output TO IThis.D64B8A7F104AF6C1;
    IThis.90008E8CE94947BC TO CT_ReactorActual.01D9354E0C07C6C2;
    IThis.FA5A2A894C4F3D58 TO StartUpDelay.DT1;
    NextFeedHorizon.25675C20D4D4E92B TO IEmergencyR1.83DE9B371B83EBB9;
    NextFeedHorizon.67679D1DCC8CE4F7 TO IEmergencyR1.5C25718B2BAE6B29;
    NextFeedHorizon.9E303FAD1787430C TO IEmergencyR2.83DE9B371B83EBB9;
    NextFeedHorizon.F5A5BE19A3003F71 TO IEmergencyR2.5C25718B2BAE6B29;
    NextFeedHorizon.4DFFB3B7D8ECCFDC TO IEmergencyR3.83DE9B371B83EBB9;
    NextFeedHorizon.9DEC5950D04DBA6C TO IEmergencyR3.5C25718B2BAE6B29;
    NextFeedHorizon.5DD234646DF00166 TO IEmergencyR4.83DE9B371B83EBB9;
    NextFeedHorizon.FB90FB87E91DB2D3 TO IEmergencyR4.5C25718B2BAE6B29;
    NextFeedHorizon.99AA9844B7E2C1B0 TO IEmergencyR5.83DE9B371B83EBB9;
    NextFeedHorizon.1B44EFA413469744 TO IEmergencyR5.5C25718B2BAE6B29;
    NextFeedHorizon.4DD7F796010A93F3 TO IEmergencyR6.83DE9B371B83EBB9;
    NextFeedHorizon.9B0B9B8D04810A81 TO IEmergencyR6.5C25718B2BAE6B29;
    FeedStarted.OUT TO FeedRun.PERMIT;
    IEmergencyR1.1D99A7E687AA4E06 TO FeedStartedSmooth.25B5287A5784F3EC;
    IEmergencyR2.1D99A7E687AA4E06 TO FeedStartedSmooth.4ABB3F1062775F74;
    IEmergencyR3.1D99A7E687AA4E06 TO FeedStartedSmooth.113D29D71E6DF4C2;
    IEmergencyR4.1D99A7E687AA4E06 TO FeedStartedSmooth.0BC4334F5BE263F8;
    IEmergencyR5.1D99A7E687AA4E06 TO FeedStartedSmooth.FB0E6D999B27FA12;
    IEmergencyR6.1D99A7E687AA4E06 TO FeedStartedSmooth.552C61FEC6B42E99;
    StartUpDelay.716D3F3042596C89 TO EmergencyReactorsControl.792E98CD16D8165F;
    EmergencyReactorsControl.93BD970A79F50FF2 TO FeedCmdTimeOutR1.C97C7F32550A1F33;
    EmergencyReactorsControl.48471A9871450B3D TO FeedCmdTimeOutR2.C97C7F32550A1F33;
    EmergencyReactorsControl.C47F108F9D450515 TO FeedCmdTimeOutR3.C97C7F32550A1F33;
    EmergencyReactorsControl.59886E5EA0464B37 TO FeedCmdTimeOutR4.C97C7F32550A1F33;
    EmergencyReactorsControl.98828EA78D316628 TO FeedCmdTimeOutR5.C97C7F32550A1F33;
    EmergencyReactorsControl.D66C5C5D632E05FA TO FeedCmdTimeOutR6.C97C7F32550A1F33;
    IEmergencyR1.1D99A7E687AA4E06 TO FeedCmdTimeOutR1.453195D0E8A9E1D1;
    IEmergencyR2.1D99A7E687AA4E06 TO FeedCmdTimeOutR2.453195D0E8A9E1D1;
    IEmergencyR3.1D99A7E687AA4E06 TO FeedCmdTimeOutR3.453195D0E8A9E1D1;
    IEmergencyR4.1D99A7E687AA4E06 TO FeedCmdTimeOutR4.453195D0E8A9E1D1;
    IEmergencyR5.1D99A7E687AA4E06 TO FeedCmdTimeOutR5.453195D0E8A9E1D1;
    IEmergencyR6.1D99A7E687AA4E06 TO FeedCmdTimeOutR6.453195D0E8A9E1D1;
    EmergencyReactorsControl.70104F20CA3ADF24 TO IEmergencyR1.B7D7393A43236C58;
    EmergencyReactorsControl.70104F20CA3ADF24 TO IEmergencyR2.B7D7393A43236C58;
    EmergencyReactorsControl.70104F20CA3ADF24 TO IEmergencyR3.B7D7393A43236C58;
    EmergencyReactorsControl.70104F20CA3ADF24 TO IEmergencyR4.B7D7393A43236C58;
    EmergencyReactorsControl.70104F20CA3ADF24 TO IEmergencyR5.B7D7393A43236C58;
    EmergencyReactorsControl.70104F20CA3ADF24 TO IEmergencyR6.B7D7393A43236C58;
    EmergencyReactorsControl.0341C3C3411D612A TO IEmergencyR1.072FACB5311A61D8;
    EmergencyReactorsControl.0341C3C3411D612A TO IEmergencyR2.072FACB5311A61D8;
    EmergencyReactorsControl.0341C3C3411D612A TO IEmergencyR3.072FACB5311A61D8;
    EmergencyReactorsControl.0341C3C3411D612A TO IEmergencyR4.072FACB5311A61D8;
    EmergencyReactorsControl.0341C3C3411D612A TO IEmergencyR5.072FACB5311A61D8;
    EmergencyReactorsControl.0341C3C3411D612A TO IEmergencyR6.072FACB5311A61D8;
    EmergencyReactorsControl.70104F20CA3ADF24 TO SD_WS2_Initialization_Manager.836EEC408BC0CBE9;
    EmergencyReactorsControl.0341C3C3411D612A TO SD_WS2_Initialization_Manager.A4F615B7B93BC654;
    SmoothEmergencyON.Output TO SD_WS2_Initialization_Manager.E8F44C2903DAE817;
    SD_WS2_Initialization_Manager.566AA45BA43174B4 TO IEmergencyR6.EEDAEC65A069032E;
    SD_WS2_Initialization_Manager.F70FEC38519C4AAA TO IEmergencyR5.EEDAEC65A069032E;
    SD_WS2_Initialization_Manager.4821ED2B62A9F30E TO IEmergencyR4.EEDAEC65A069032E;
    SD_WS2_Initialization_Manager.17646700D696E2B5 TO IEmergencyR3.EEDAEC65A069032E;
    SD_WS2_Initialization_Manager.234E3C02BCC1EECC TO IEmergencyR1.EEDAEC65A069032E;
    SD_WS2_Initialization_Manager.DDCC6CFA75DFB7EF TO IEmergencyR2.EEDAEC65A069032E;
    IEmergencyR1.613E286D19768818 TO SD_WS2_Initialization_Manager.AA9C2322755234D4;
    IEmergencyR2.613E286D19768818 TO SD_WS2_Initialization_Manager.3AAB6E0EA8D414C3;
    IEmergencyR3.613E286D19768818 TO SD_WS2_Initialization_Manager.142729A22C77C117;
    IEmergencyR4.613E286D19768818 TO SD_WS2_Initialization_Manager.AFD64E411479B55C;
    IEmergencyR5.613E286D19768818 TO SD_WS2_Initialization_Manager.37E13E80A15F0DC1;
    IEmergencyR6.613E286D19768818 TO SD_WS2_Initialization_Manager.7D37330759993BBA;
    IEmergencyR1.B3BCA5E1F4B3D013 TO SD_WS2_Initialization_Manager.D2A6AD247A4FAA4E;
    IEmergencyR2.B3BCA5E1F4B3D013 TO SD_WS2_Initialization_Manager.F643778FAE08D711;
    IEmergencyR3.B3BCA5E1F4B3D013 TO SD_WS2_Initialization_Manager.846CE7FC989F43EC;
    Delay.716D3F3042596C89 TO SD_WS2_Initialization_Manager.8F677304EBF56E28;
    SmoothEmergencyON.Output TO StartFeedPosition.50516E5FA0A93F3A;
    SmoothNumberOfReactors2.A6DEF5F9C27C1848 TO StartFeedPosition.6C5BFBC6FB7FAD46;
    NumberOfReactorsAv3.A6DEF5F9C27C1848 TO StartFeedPosition.9FD4887EB6BF3EFF;
    FeedStartedSmooth.AA81B8787A42C5C8 TO FeedStarted.IN1;
    FeedStartedSmooth.9956B7B3B3929CFE TO FeedStarted.IN2;
    FeedStartedSmooth.0578107E6CFA5800 TO FeedStarted.IN3;
    FeedStartedSmooth.167BD6731FEB1D53 TO FeedStarted.IN4;
    FeedStartedSmooth.1AB852B2890146E4 TO FeedStarted.IN5;
    FeedStartedSmooth.6C1C82B2CFBF666D TO FeedStarted.IN6;
    IReactor1.3C69BB1A066E9338 TO ReactorAvaibilityChanged.25B5287A5784F3EC;
    IReactor2.3C69BB1A066E9338 TO ReactorAvaibilityChanged.4ABB3F1062775F74;
    IReactor3.3C69BB1A066E9338 TO ReactorAvaibilityChanged.113D29D71E6DF4C2;
    IReactor4.3C69BB1A066E9338 TO ReactorAvaibilityChanged.0BC4334F5BE263F8;
    IReactor5.3C69BB1A066E9338 TO ReactorAvaibilityChanged.FB0E6D999B27FA12;
    IReactor6.3C69BB1A066E9338 TO ReactorAvaibilityChanged.552C61FEC6B42E99;
    SmoothEmergencyON.Output TO EmergencyONPermit.PERMIT;
    ReactorAvaibilityChanged.AA81B8787A42C5C8 TO RxNoAvThenRxAv.1132AFD18E56345D;
    ReactorAvaibilityChanged.9956B7B3B3929CFE TO RxNoAvThenRxAv.6C59961ACF104AA7;
    ReactorAvaibilityChanged.0578107E6CFA5800 TO RxNoAvThenRxAv.BF70B6C486B5373C;
    SmoothEmergencyON.Output TO RxNoAvThenRxAv.088CD67AD55F3330;
    RxNoAvThenRxAv.EC29A541E7FBE6C9 TO IEmergencyR1.713BAA92BE7C280E;
    RxNoAvThenRxAv.F577B5E8F808E26B TO IEmergencyR2.713BAA92BE7C280E;
    RxNoAvThenRxAv.403B70773A4F56EF TO IEmergencyR3.713BAA92BE7C280E;
    RxNoAvThenRxAv.F047C6A8D1E626BD TO IEmergencyR4.713BAA92BE7C280E;
    RxNoAvThenRxAv.FA7EB0D9886C53C5 TO IEmergencyR5.713BAA92BE7C280E;
    RxNoAvThenRxAv.3C16CC1F05F5D6CE TO IEmergencyR6.713BAA92BE7C280E;
    ISludgeBuffer.3C69BB1A066E9338 TO IEmergencyR1.1675BB23EEFCF5E9;
    ISludgeBuffer.3C69BB1A066E9338 TO IEmergencyR2.1675BB23EEFCF5E9;
    ISludgeBuffer.3C69BB1A066E9338 TO IEmergencyR4.1675BB23EEFCF5E9;
    ISludgeBuffer.3C69BB1A066E9338 TO IEmergencyR3.1675BB23EEFCF5E9;
    ISludgeBuffer.3C69BB1A066E9338 TO IEmergencyR5.1675BB23EEFCF5E9;
    ISludgeBuffer.3C69BB1A066E9338 TO IEmergencyR6.1675BB23EEFCF5E9;
  END_CONNECTIONS
END_FUNCTION_BLOCK
